{attribute 'pack_mode' := '1'} 
TYPE ST_AxisTableBuf :
STRUCT
	Table	: ARRAY [1..No, 0..1999] OF LREAL;
	OK		: BOOL;
END_STRUCT
END_TYPE

(* stored: Version 1.1.0.1, ProductVersion 3.1.4024.9
   DUT ST_AxisTableBuf: Id {573478b2-28b8-40ad-b94d-cef3abcefc96} *)
